// TwinCAT 3 PLC project TcAbbLinkin
// ProgramVersion: 3.1.4024.0
// libraries:
//   Tc2_Standard, * (Beckhoff Automation GmbH)
//   Tc2_System, * (Beckhoff Automation GmbH)
//   Tc3_Module, * (Beckhoff Automation GmbH)
// project tree:
//   / PlcTask.TcTTO
//   POUs/ MAIN.TcPOU, TcAbbLinkin.TcPOU

CONFIGURATION TcAbbLinkin
    RESOURCE PLC ON TwinCAT3
        TASK PlcTask(INTERVAL := T#10ms, PRIORITY := 20);
        PROGRAM MAIN WITH PlcTask : MAIN;
    END_RESOURCE
END_CONFIGURATION

// ---- POUs/MAIN.TcPOU
PROGRAM MAIN
VAR
	myrobot: 	TcAbbLinkin;
	hmiPowerOn: BOOL;
	isPowered: INT;
	state: INT;
	the: INT;
	seq:	asdf;
	mycommand: 	PLCOpenCall;
END_VAR



myRobot();



IF (hmiPowerOn) THEN
	myrobot.RobotPowerOn();
	
	
	
	
	hmiPowerOn := FALSE;
END_IF


IF myrobot.isPowered() THEN
	alarm("robot is powered");
END_IF


myrobot.GetState();

CASE state OF 
	
	1: 
		
		myrobot.RobotPowerOn();
	
		state := 2;
	2:
		//IF myrobot.isPowered() THEN
		IF myrobot.powered THEN
			state := 3;
		END_IF

	3: 


END_CASE


CASE seq.doState() OF 
	
	1: 
		IF seq.onEntry() THEN
			myrobot.RobotPowerOn(seq);
		END_IF
		
		seq.onSuccess(2);
	2:
		//IF myrobot.isPowered() THEN
		IF myrobot.powered THEN
			state := 3;
		END_IF

	3: 


END_CASE



IF localCmd THEN
	myrobot.RobotPowerOn(mycommand);
END_IF


IF mycommand.Done OR mycommand.Error THEN
	alarm();
END_IF

END_PROGRAM

// ---- POUs/TcAbbLinkin.TcPOU
FUNCTION_BLOCK TcAbbLinkin
VAR_INPUT
END_VAR
VAR_OUTPUT
END_VAR
VAR
	powerCommand: PLCOpenCommand;
END_VAR



IF powerCommand.Consume THEN
	
	// run through state
	
	
END_IF


// When power command is done
IF robotIspowered THEN
	
	powerCommand.Finish()

END_IF

METHOD ConnectionReset : BOOL
VAR_INPUT
END_VAR
END_METHOD

METHOD ConnectionSetup : BOOL
VAR_INPUT
END_VAR
END_METHOD

METHOD GetIO : BOOL
VAR_INPUT
END_VAR
END_METHOD

METHOD GetState : BOOL
VAR_INPUT
END_VAR
END_METHOD

METHOD GetSymbol : BOOL
VAR_INPUT
END_VAR
END_METHOD

METHOD IOWatchInit : BOOL
VAR_INPUT
END_VAR
END_METHOD

METHOD RapidReset : BOOL
VAR_INPUT
END_VAR
END_METHOD

METHOD RobotMotorsOff : BOOL
VAR_INPUT
END_VAR
END_METHOD

METHOD RobotMotorsOn : BOOL
VAR_INPUT
END_VAR
END_METHOD

METHOD RobotPowerOff : BOOL
VAR_INPUT
END_VAR
END_METHOD

METHOD RobotPowerOn : BOOL
VAR_INPUT
	status: IPLCOpenCommand;
END_VAR

IF status <> 0 THEN
	status.Start(powerCommand);
ELSE
	powerCommand.Execute := TRUE;
END_IF
END_METHOD

METHOD RobotStart : BOOL
VAR_INPUT
END_VAR
END_METHOD

METHOD RobotStop : BOOL
VAR_INPUT
END_VAR
END_METHOD

METHOD SetIO : BOOL
VAR_INPUT
END_VAR
END_METHOD

METHOD SetSymbol : BOOL
VAR_INPUT
END_VAR
END_METHOD

END_FUNCTION_BLOCK
